RoboDK station: SpiralMeca.rdk

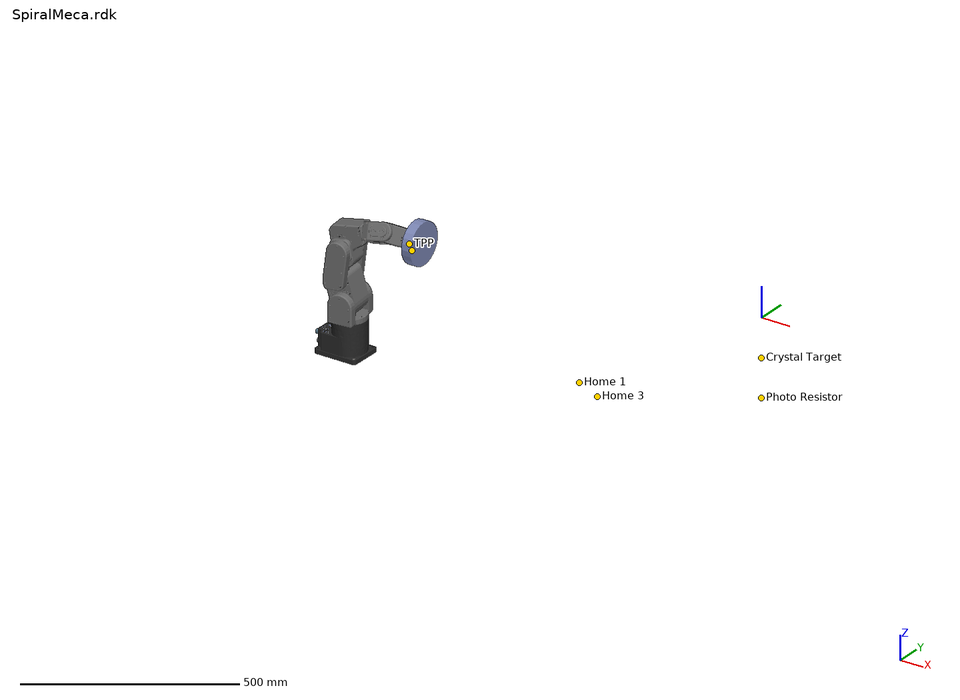
[picture v0: the station drawn from its stored meshes, robots at their saved joint values, targets as dots, program paths as lines]
Station SpiralMeca (saved by RoboDK 5.5.2). Poses are relative to the parent item; angles as X-Y-Z fixed-axis rotations.
  - robot Mecademic Meca500 R3: 6 axes
      modified DH rows (alpha deg, a mm, theta deg, d mm): 0, 0, 0, 135; -90, 0, -90, 0; 0, 135, 0, 0; -90, 38, 0, 120; 90, 0, 0, 0; -90, 0, 180, 70
      joint limits [-150, -70, -135, -170, -115, -720] to [150, 90, 70, 170, 115, 720]; home [0, 0, 0, 0, 0, 0]; saved at [5.545, -3.441, -6.55, -29.231, 11.413, 28.746]
    - tool CrystalToolSample, TCP at (0, 0, 0) mm, size 107.9 x 25.4 x 107.9 mm, geometry from CrystalToolSample.STEP
  - frame LED at (1143, 0, 409.6) mm
    - target TPP (Cartesian target) at (-970, -10, -81.6) mm, rotated rx 0 ry 90 rz 0 deg; joints [-5.545, -3.441, -6.55, 29.231, 11.413, -28.746] of Mecademic Meca500 R3
    - target Home 3 (Cartesian target) at (245.4, -1000, 268) mm, rotated rx 0 ry 90 rz 0 deg; joints [0, 10.295, 7.197, 0, -17.492, 0] of Mecademic Meca500 R3
    - target Home 1 (joint target) at (215.4, -1030, 308) mm, rotated rx 0 ry 90 rz 0 deg; joints [0, 0, 0, 0, 0, 0] of Mecademic Meca500 R3
    - target Target 47 (joint target) at (342.4, -1030, 308) mm, rotated rx 0 ry 90 rz 0 deg; joints [0, 11.211, -12.445, 0, 1.234, 0] of Mecademic Meca500 R3
    - target Photo Resistor (Cartesian target) at (0, 0, -203.2) mm; joints [0, 0, 0, 0, 0, 0] of Mecademic Meca500 R3
    - target Crystal Target (Cartesian target) at (0, 0, -101.6) mm; joints [-23.128, -26.053, 31.636, -77.168, -23.756, 166.237] of Mecademic Meca500 R3
    - target Target 7 (Cartesian target) at (-970.2, 0, -101.6) mm, rotated rx 0 ry 90 rz 0 deg; joints [0, -22.455, 17.494, 0, 4.961, 0] of Mecademic Meca500 R3
    - target Target 8 (Cartesian target) at (-970.2, 0, -101.6) mm, rotated rx 0 ry 90 rz 0 deg; joints [0, -33.951, 22.527, 0, 11.424, 0] of Mecademic Meca500 R3
  - Python program Spiral (listed below)
  - Python program Go Home (listed below)
  - Python program TEST SSAP (listed below)
  - Python program Prog4 (listed below)
  - Python program Linear Move (listed below)
  - Python program SSAP (listed below)
    - Python program Test SSAP 2 (listed below)
    - Python program Test SSAP 3 (listed below)
    - Python program Smart Spiral SSAP (listed below)
  - Python program Set Target Pos (listed below)
  - Python program Hexagon Test (listed below)
  - Python program Prog12 (listed below)
  - Python program Prog13 (listed below)

--- Python program Spiral ---
"""
Created on Thu Jan 19 18:43:18 2023

@author: westj
"""
from robodk.robolink import *       # import the robolink library (bridge with RoboDK)
RDK = Robolink()
from robodk.robomath import *
import math
import numpy as np
import matplotlib.pyplot as plt

class Spiral:
    def __init__(self,x0:float,y0:float,points:float) -> None:
        self.x0=x0 #x offset
        self.y0=y0 #y offset
        self.points=points

    def build(self, radius:float, spacing:float):
        revs=radius/spacing            #calc number of revolutions
        k=spacing/(2*np.pi)
        theta=np.array(np.linspace(0,revs*2*np.pi,self.points)) #how many points and angle coord
        r=k * theta                       #radius coord
        x=(r*np.cos(theta)+self.x0)
        y=(r*np.sin(theta)+self.y0)             #convert to y cartesian

        return x, y #convert to x cartesian


if __name__=="__main__":
    print('Calling spiral from class')
    R=30
    S=10
    TSpeed=10
    cur_spiral=Spiral(0,0,500)
    x,y=cur_spiral.build(R,S)


 #   print(cur_spiral.build(R,S))
  #  plt.plot(x, y, color = 'red', marker = "o")
  #  plt.axis('equal')
  #  plt.show()

#______Robot Movement_________________________________________

robot = RDK.Item('Mecademic Meca500 R3')
home = RDK.Item('Home 1')
target = RDK.Item('Target 2')# retrieve the Target item


robot.MoveJ(home)

robot.MoveJ(target)                 # move the robot to the target
#for i in x:
    #robot.MoveL(target.Pose()*transl(coord))

for i in range(len(x)):

    coord=(x[i],y[i],0)
    robot.MoveJ(target.Pose()*transl(coord))
    robot.WaitFinished()
    #print(coord)
    #print('')

--- Python program Go Home ---
# Type help("robodk.robolink") or help("robodk.robomath") for more information
# Press F5 to run the script
# Documentation: https://robodk.com/doc/en/RoboDK-API.html
# Reference:     https://robodk.com/doc/en/PythonAPI/robodk.html
# Note: It is not required to keep a copy of this file, your Python script is saved with your RDK project

# You can also use the new version of the API:
from robodk import robolink    # RoboDK API
from robodk import robomath    # Robot toolbox
RDK = robolink.Robolink()

robot = RDK.Item('Mecademic Meca500 R3')
home = RDK.Item('Home 1')
robot.MoveJ(home)

--- Python program TEST SSAP ---
"""
Created on Thu Jan 19 18:43:18 2023

@author: westj
"""
from robodk.robolink import *       # import the robolink library (bridge with RoboDK)
RDK = Robolink()
from robodk.robomath import *
import math
import numpy as np
import matplotlib.pyplot as plt
import array
import pandas as pd
from scipy.signal import find_peaks
from scipy.stats import linregress

class Spiral:
    def __init__(self,x0:float,y0:float,points:float) -> None:
        self.x0=x0 #x offset
        self.y0=y0 #y offset
        self.points=points

    def build(self, radius:float, spacing:float):
        revs=radius/spacing            #calc number of revolutions
        k=spacing/(2*np.pi)
        theta=np.array(np.linspace(0,revs*2*np.pi,self.points)) #how many points and angle coord
        r=k * theta                       #radius coord
        x=(r*np.cos(theta)+self.x0)       #convert to x cartesian
        y=(r*np.sin(theta)+self.y0)       #convert to y cartesian

        return x, y

class Linear:
    def __init__(self,data,points):
        self.data=data #data
        self.points=points #x offset

    def get(self,x):
        peaks= find_peaks(self.data['Intensity'], height=.1)

        H=peaks[1]['peak_heights']
        A=[]
        for i in range(len(IPeaks)):
            corr=[IPeaks[i],H[i]]
            A.append(corr)
        SA=sorted(A, key=lambda x: x[1], reverse=True) #sort by peak height largest to smallest
        print(SA)
        XPP=[]
        YPP=[]
        for i in range(self.points):
            #ICP.append(SA[i][0])
            XPP.append(self.data['X'][SA[i][0]])
            YPP.append(self.data['Y'][SA[i][0]])
        LRR=linregress(XPP,YPP)

        return LRR[0]*x+LRR[1]


class Intensity: #intensity function is a gaussian curve
    def __init__(self,x0:float,y0:float, mu_x, mu_y, sigma_x, sigma_y):
        self.x0=-x0 #x offset
        self.y0=-y0 #y offset
        self.mu_x=mu_x
        self.mu_y=mu_y
        self.sigma_x=sigma_x #x squish/stretch
        self.sigma_y=sigma_y #y sqush/stretch


    def get(self,x, y): #gaussian curve definition
        I=np.exp(-0.5 * (((x +self.x0- self.mu_x) / self.sigma_x)**2 + ((y+self.y0 - self.mu_y) / self.sigma_y)**2))
        return I


#*****************************************************************************************************************
#___Initialization______________
xl=0
yl=0
Loops=3
robot = RDK.Item('Mecademic Meca500 R3')
home = RDK.Item('Home 1')
target = RDK.Item('Target 2')# retrieve the Target item

robot.MoveJ(home)
robot.MoveJ(target)



for L in range(1,Loops+1):
    print(L)
    if __name__=="__main__":
        print('Calling spiral from class')

        cur_spiral=Spiral(xl,yl,200) #setting params of the spiral we will be using
        x,y=cur_spiral.build(10/L**L,5/L) #build our spiral x y coords
        Ix=1.24
        Iy=-2.3
        TestInt=Intensity(Ix,Iy,0,0,10,10) #set test intensity parameters

        #Plot our spiral
        # plt.plot(x, y, color = 'red', marker = "o")
        # plt.axis('equal')
        # plt.show()

    #initialize params
    X=[]
    Y=[]
    Z=[]
    Iv=[]
    Cv=[]

    for i in range(len(x)): #loop to get coord and corresponding intensity
        coord=(x[i],y[i],0)
        X.append(x[i])
        Y.append(y[i])
        Z.append(0)
        Ic=TestInt.get(x[i],y[i])
        Iv.append(np.array(Ic))

        robot.MoveJ(target.Pose()*transl(coord))
        robot.WaitFinished()
        #pandas dictionary
        titled_columns={'X': X,'Y': Y,'Z': Z,
                        'Intensity': Iv}
        data = pd.DataFrame(titled_columns)


    peaks= find_peaks(data['Intensity'], height=.1)
    IPeaks=peaks[0]
    H=peaks[1]['peak_heights']
    A=[]
    for i in range(len(IPeaks)):
        corr=[IPeaks[i],H[i]]
        A.append(corr)



    SA=sorted(A, key=lambda x: x[1], reverse=True) #sort by peak height largest to smallest
    if len(SA) == 1:
        print('one peak detected')
        break
    else:

     CL=Linear(data,2) #current linear line definition

    step=.1/L #linear step size
    xl=data['X'][SA[0][0]] #start x
    yl=CL.get(xl) #start y

    Xl=[xl]
    Yl=[yl]
    Il=[TestInt.get(xl,yl)]

    if  data['X'][SA[0][0]] < data['X'][SA[1][0]]:
        step=step
    else:
        step=-step


    while TestInt.get(xl+step,CL.get(xl+step)) >= TestInt.get(xl,CL.get(xl)):

        xl=xl+step
        yl=CL.get(xl)
        il=TestInt.get(xl,yl)
        Xl.append(xl)
        Yl.append(yl)
        Il.append(il)
        coord=(xl,yl,0)
        robot.MoveJ(target.Pose()*transl(coord))



    LLdata={'X':Xl,'Y':Yl,'I':Il}
    Ldata=pd.DataFrame(LLdata)

    fig = plt.figure()
    plt.style.use('seaborn-notebook')
    ax = fig.add_subplot(111, projection='3d')
    ax.plot3D(data['X'], data['Y'], data['Intensity'])
    ax.plot3D(data['X'][IPeaks], data['Y'][IPeaks], data['Intensity'][IPeaks],"x")
    ax.plot3D(Xl, Yl, Il,'o')

    ax.set_xlabel('X axis')
    ax.set_ylabel('Y axis')
    ax.set_zlabel('Z axis')
plt.show()




E=np.sqrt((Ix-xl)**2+(Iy-yl)**2)
print('***Linear Translation********************************************************')
print(Ldata)
print('_________SSAP Report:_________')
print('Calculated peak is at',xl,yl)
print('True peak is at',Ix,Iy)
print('Error is:',E)
print('Linear step size is:',step)

--- Python program Prog4 ---
# -*- coding: utf-8 -*-
"""
Created on Tue Feb 14 10:13:50 2023

@author: ChatGPT/ Jeremy West
"""

import math
from robodk.robolink import *
from robodk import robomath
RDK = Robolink()

target = RDK.Item('Target 2')# retrieve the Target item
robot = RDK.Item('Mecademic Meca500 R3')

# Define the position of the robot's tool
x = 100
y = 100
z = 300

# Define the orientation of the robot's tool using Euler angles (in degrees)
a = 0   # rotation around x-axis
b = 0    # rotation around y-axis
g = 0    # rotation around z-axis


# Set the robot's tool pose to the defined pose
#robodk.robomath.TxyzRxyz_2_Pose(xyzrpw) #[x,y,z,a,b,g]

#pose=robodk.robomath.Pose([x,y,z,a,b,g])
robot.setJoints([0,0,0,0,0,0])
robot.MoveJ(target)
approach = target.Pose()*transl(0,0,-100)
robot.MoveL(approach)

#print(pose)


robot.setPose(pose)

--- Python program Linear Move ---
from robodk.robolink import *       # import the robolink library (bridge with RoboDK)
from robodk.robomath import *       # import the robotics toolbox
RDK = Robolink()                    # establish a link with the simulator
robot = RDK.Item('Mecademic Meca500 R3')     # retrieve the robot by name


robot.setSpeed(100)  # Set linear speed in mm/s
robot.setJoints([0,0,0,0,0,0])      # set all robot axes to zero

tool=RDK.Item('CrystalToolSample')
robot.setPoseTool(tool) # Update the TCP

target = RDK.Item('TPP')         # retrieve the Target item
robot.MoveJ(target)                 # move the robot to the target


Final = target.Pose()*transl(0,20,0)
print(target.Pose())

rj=robot.Joints()

print(robot.MoveL_Test(rj,Final))

if robot.MoveL_Test(rj,Final) == 0:         # linear move to the approach position
    robot.MoveL(Final)


print('approach reached')
print('Attempting pose', Final)
#robot.MoveL(pose)

--- Python program SSAP ---
"""
Created on Thu Jan 19 18:43:18 2023

@author: westj
"""
from robodk.robolink import *       # import the robolink library (bridge with RoboDK)
RDK = Robolink()
from robodk.robomath import *
import math
import numpy as np
import matplotlib.pyplot as plt
import array
import pandas as pd
import requests
import re
from scipy.signal import find_peaks
from scipy.stats import linregress

class Spiral:
    def __init__(self,x0:float,y0:float,points:float) -> None:
        self.x0=x0 #x offset
        self.y0=y0 #y offset
        self.points=points

    def build(self, radius:float, spacing:float):
        revs=radius/spacing            #calc number of revolutions
        k=spacing/(2*np.pi)
        theta=np.array(np.linspace(0,revs*2*np.pi,self.points)) #how many points and angle coord
        r=k * theta                       #radius coord
        x=(r*np.cos(theta)+self.x0)       #convert to x cartesian
        y=(r*np.sin(theta)+self.y0)       #convert to y cartesian

        return x, y

class Linear:
    def __init__(self,data,points):
        self.data=data #data
        self.points=points #x offset

    def get(self,x):
        peaks= find_peaks(self.data['Intensity'], height=-900)

        H=peaks[1]['peak_heights']
        A=[]
        for i in range(len(IPeaks)):
            corr=[IPeaks[i],H[i]]
            A.append(corr)
        SA=sorted(A, key=lambda x: x[1], reverse=True) #sort by peak height largest to smallest
        print(SA)
        XPP=[]
        YPP=[]
        for i in range(self.points):
            #ICP.append(SA[i][0])
            XPP.append(self.data['X'][SA[i][0]])
            YPP.append(self.data['Y'][SA[i][0]])
        LRR=linregress(XPP,YPP)

        return LRR[0]*x+LRR[1]


class Intensity: #intensity function is a gaussian curve
    def __init__(self,x0:float,y0:float, mu_x, mu_y, sigma_x, sigma_y):
        self.x0=-x0 #x offset
        self.y0=-y0 #y offset
        self.mu_x=mu_x
        self.mu_y=mu_y
        self.sigma_x=sigma_x #x squish/stretch
        self.sigma_y=sigma_y #y sqush/stretch


    def get(self,x, y): #gaussian curve definition
        I=np.exp(-0.5 * (((x +self.x0- self.mu_x) / self.sigma_x)**2 + ((y+self.y0 - self.mu_y) / self.sigma_y)**2))
        return I

class Photoresistor:
    def __init__(self,url) -> None:
        self.url=url
    def get(self):
        response = requests.get(self.url)
        if response.ok:
            value = response.text
            pr=re.findall(r'\d+',value)
            pri=-int(pr[0])
            #print('Received value:', value)
            #print('Number', PR)
        else:
            print('Error:', response.status_code)


        return pri


#*****************************************************************************************************************
#___Initialization______________
xl=0
yl=0
Loops=3
robot = RDK.Item('Mecademic Meca500 R3')
home = RDK.Item('Home 1')
target = RDK.Item('Target 2')# retrieve the Target item
PR=Photoresistor( 'http://192.168.0.24')

robot.MoveJ(home)
robot.MoveJ(target)



for L in range(1,Loops+1):
    print(L)
    if __name__=="__main__":
        print('Calling spiral from class')

        cur_spiral=Spiral(xl,yl,200) #setting params of the spiral we will be using
        x,y=cur_spiral.build(30/L**L,5/L) #build our spiral x y coords
        Ix=1.24
        Iy=-2.3
        TestInt=Intensity(Ix,Iy,0,0,10,10) #set test intensity parameters

        #Plot our spiral
        # plt.plot(x, y, color = 'red', marker = "o")
        # plt.axis('equal')
        # plt.show()

    #initialize params
    X=[]
    Y=[]
    Z=[]
    Iv=[]
    Cv=[]

    for i in range(len(x)): #loop to get coord and corresponding intensity
        coord=(x[i],y[i],0)
        X.append(x[i])
        Y.append(y[i])
        Z.append(0)
        Ic=PR.get()

        Iv.append(np.array(Ic))

        robot.MoveJ(target.Pose()*transl(coord))
        robot.WaitFinished()
        #pandas dictionary
        titled_columns={'X': X,'Y': Y,'Z': Z,
                        'Intensity': Iv}
        data = pd.DataFrame(titled_columns)


    peaks= find_peaks(data['Intensity'], height=-900)
    print('peaks',peaks)


    IPeaks=peaks[0]
    H=peaks[1]['peak_heights']
    A=[]
    for i in range(len(IPeaks)):
        corr=[IPeaks[i],H[i]]

        A.append(corr)



    SA=sorted(A, key=lambda x: x[1], reverse=True) #sort by peak height largest to smallest
    if len(SA) == 1:
        print('one peak detected')
        break
    else:

     CL=Linear(data,2) #current linear line definition

    step=.1/L #linear step size
    xl=data['X'][SA[0][0]] #start x
    yl=CL.get(xl) #start y

    Xl=[xl]
    Yl=[yl]
    PRS=SA[0][1]
    Il=[PRS]

    if  data['X'][SA[0][0]] < data['X'][SA[1][0]]:
        step=step
    else:
        step=-step


    while PR.get() >= .99*PRS:

        xl=xl+step
        yl=CL.get(xl)
        PRS=PR.get()
        Xl.append(xl)
        Yl.append(yl)
        Il.append(PRS)
        coord=(xl,yl,0)
        robot.MoveJ(target.Pose()*transl(coord))



    LLdata={'X':Xl,'Y':Yl,'I':Il}
    Ldata=pd.DataFrame(LLdata)

    fig = plt.figure()
    plt.style.use('seaborn-notebook')
    ax = fig.add_subplot(111, projection='3d')
    ax.plot3D(data['X'], data['Y'], data['Intensity'])
    ax.plot3D(data['X'][IPeaks], data['Y'][IPeaks], data['Intensity'][IPeaks],"x")
    ax.plot3D(Xl, Yl, Il,'o')

    ax.set_xlabel('X axis')
    ax.set_ylabel('Y axis')
    ax.set_zlabel('Z axis')
plt.show()




E=np.sqrt((Ix-xl)**2+(Iy-yl)**2)
print('***Linear Translation********************************************************')
print(Ldata)
print('_________SSAP Report:_________')
print('Calculated peak is at',xl,yl)
print('True peak is at',Ix,Iy)
print('Error is:',E)
print('Linear step size is:',step)

--- Python program Test SSAP 2 ---
"""
Created on Thu Jan 19 18:43:18 2023

@author: westj
"""
from robodk.robolink import *       # import the robolink library (bridge with RoboDK)
RDK = Robolink()
from robodk.robomath import *
import math
import numpy as np
import matplotlib.pyplot as plt
import array
import pandas as pd
import requests
import re
from scipy.signal import find_peaks
from scipy.stats import linregress
#******CLASSES AND CLASS FUNCTIONS****************************************************************************
class Spiral:
    def __init__(self,x0:float,y0:float,points:float) -> None:
        self.x0=x0 #x offset
        self.y0=y0 #y offset
        self.points=points

    def build(self, radius:float, spacing:float):
        revs=radius/spacing            #calc number of revolutions
        k=spacing/(2*np.pi)
        theta=np.array(np.linspace(0,revs*2*np.pi,self.points)) #how many points and angle coord
        r=k * theta                       #radius coord
        x=(r*np.cos(theta)+self.x0)       #convert to x cartesian
        y=(r*np.sin(theta)+self.y0)       #convert to y cartesian
        return x, y

class Linear:
    def __init__(self,data,points):
        self.data=data #data
        self.points=points #x offset

    def get(self,x):
        peaks= find_peaks(self.data['Intensity'], height=-900)
        IPeaks=peaks[0]
        H=peaks[1]['peak_heights']
        A=[]
        for i in range(len(IPeaks)):
            corr=[IPeaks[i],H[i]]
            A.append(corr)
        SA=sorted(A, key=lambda x: x[1], reverse=True) #sort by peak height largest to smallest
        if len(SA) <= 1:

            E=np.sqrt((Ix-xl)**2+(Iy-yl)**2)
            print('***Linear Translation********************************************************')
            print(Ldata)
            print('_________SSAP Report:_________')
            print('Calculated peak is at',xl,yl)
            print('True peak is at',Ix,Iy)
            print('Error is:',E)
            print('Linear step size is:',step)
            raise Exception("Spiral did not find enough peaks")
        XPP=[]
        YPP=[]
        for i in range(self.points):
            #ICP.append(SA[i][0])
            XPP.append(self.data['X'][SA[i][0]])
            YPP.append(self.data['Y'][SA[i][0]])
        LRR=linregress(XPP,YPP)

        return LRR[0]*x+LRR[1]

    def getSA(self):
        peaks= find_peaks(self.data['Intensity'], height=-900)
        IPeaks=peaks[0]
        H=peaks[1]['peak_heights']
        A=[]
        for i in range(len(IPeaks)):
            corr=[IPeaks[i],H[i]]
            A.append(corr)
        SA=sorted(A, key=lambda g: g[1], reverse=True) #sort by peak height largest to smallest
        return SA,IPeaks

class Intensity: #intensity function is a gaussian curve
    def __init__(self,x0:float,y0:float, mu_x, mu_y, sigma_x, sigma_y):
        self.x0=-x0 #x offset
        self.y0=-y0 #y offset
        self.mu_x=mu_x
        self.mu_y=mu_y
        self.sigma_x=sigma_x #x squish/stretch
        self.sigma_y=sigma_y #y sqush/stretch


    def get(self,x, y): #gaussian curve definition
        I=np.exp(-0.5 * (((x +self.x0- self.mu_x) / self.sigma_x)**2 + ((y+self.y0 - self.mu_y) / self.sigma_y)**2))
        return I

class Photoresistor:
    def __init__(self,url) -> None:
        self.url=url
    def get(self):
        response = requests.get(self.url)
        if response.ok:
            value = response.text
            pr=re.findall(r'\d+',value)
            pri=-int(pr[0])
            #print('Received value:', value)
            #print('Number', PR)
        else:
            print('Error:', response.status_code)


        return pri


#***SPIRAL SCANNING ALIGNMENT PROCEDURE**************************************************************************************************************
#___Initialization______________
xl=0 #starting offset from target for spiral
yl=0
Loops=2 #number of loops to run SSAP

robot = RDK.Item('Mecademic Meca500 R3') #define robot
home = RDK.Item('Home 1') #define robot home
target = RDK.Item('Target 2')# retrieve the Target item
PR=Photoresistor( 'http://192.168.0.24') #Photoresistor webserver IP

robot.MoveJ(home)
print('Robot homed')
robot.MoveJ(target)
print('Robot target approached')

for L in range(1,Loops+1):
    if __name__=="__main__":
        print('Starting Spiral '+str(L))

        cur_spiral=Spiral(xl,yl,200) #setting params of the spiral we will be using
        x,y=cur_spiral.build(20/L**L,3/L) #build our spiral x y coords
        Ix=-15.24
        Iy=25.3
        TestInt=Intensity(Ix,Iy,0,0,10,10) #set test intensity parameters

        #Plot our spiral
        # plt.plot(x, y, color = 'red', marker = "o")
        # plt.axis('equal')
        # plt.show()

    #initialize params
    X=[]
    Y=[]
    Z=[]
    Iv=[]
    Cv=[]

    for i in range(len(x)): #loop to get coord and corresponding intensity
        coord=(x[i],y[i],0)
        X.append(x[i])
        Y.append(y[i])
        Z.append(0)
        #Ic=PR.get() #get intensity for PR for online run
        Ic=TestInt.get(x[i],y[i]) #test intensity get
        Iv.append(np.array(Ic))

        robot.MoveJ(target.Pose()*transl(coord))
        robot.WaitFinished()

        #pandas dictionary
        titled_columns={'X': X,'Y': Y,'Z': Z,
                        'Intensity': Iv}
        data = pd.DataFrame(titled_columns)

    print('Spiral ' +str(L)+ ' Completed')

    CL=Linear(data,2) #current linear line definition
    SA,IPeaks=CL.getSA()

    step=.1/L #linear step size
    xl=data['X'][SA[0][0]] #start x
    yl=CL.get(xl) #start y

    Xl=[xl,xl,xl]
    Yl=[yl,yl,yl]
    PRS=SA[0][1]
    Il=[PRS,PRS,PRS]
    ave_c=3 #number of intetensity terms to average
    IAv=np.average(Il[:ave_c])

    if  data['X'][SA[0][0]] < data['X'][SA[1][0]]:  #find direction to move based on location of next highest intensity
        step=-step
    else:
        step=step

    print('Linear move '+str(L)+ ': STARTED')
    while PRS >= .99*IAv:
        IAv=np.average(Il[:ave_c])
        xl=xl+step
        yl=CL.get(xl)
        #PRS=PR.get()
        PRS=TestInt.get(xl,yl)
        Xl.append(xl)
        Yl.append(yl)
        Il.append(PRS)
        coord=(xl,yl,0)
        robot.MoveJ(target.Pose()*transl(coord))
    print('Linear move '+str(L)+ ': COMPLETED')

    LLdata={'X':Xl,'Y':Yl,'I':Il}
    Ldata=pd.DataFrame(LLdata)

    Lmax_I=Il.index(max(Ldata['I']))
    xl=Xl[Lmax_I]
    yl=Yl[Lmax_I]

    fig = plt.figure()
    #plt.style.use('seaborn-notebook')
    ax = fig.add_subplot(111, projection='3d')
    ax.plot3D(data['X'], data['Y'], data['Intensity'])
    ax.plot3D(data['X'][IPeaks], data['Y'][IPeaks], data['Intensity'][IPeaks],"x")
    ax.plot3D(xl, yl, max(Ldata['I']),"x")
    ax.plot3D(Xl, Yl, Il,'o')

    ax.set_xlabel('X axis')
    ax.set_ylabel('Y axis')
    ax.set_zlabel('Z axis')
plt.show()




E=np.sqrt((Ix-xl)**2+(Iy-yl)**2)
print('***Linear Translation********************************************************')
print(Ldata)
print('_________SSAP Report:_________')
print('Calculated peak is at',xl,yl)
print('True peak is at',Ix,Iy)
print('Error is:',E)
print('Linear step size is:',step)

--- Python program Test SSAP 3 ---
"""
Created on Thu Jan 19 18:43:18 2023

@author: westj
"""
from robodk.robolink import *       # import the robolink library (bridge with RoboDK)
RDK = Robolink()
from robodk.robomath import *
import math
import numpy as np
import matplotlib.pyplot as plt
import array
import pandas as pd
import requests
import re
from scipy.signal import find_peaks, peak_prominences
from scipy.stats import linregress
#******CLASSES AND CLASS FUNCTIONS****************************************************************************
class Spiral:
    def __init__(self,x0:float,y0:float,points:float) -> None:
        self.x0=x0 #x offset
        self.y0=y0 #y offset
        self.points=points

    def build(self, radius:float, spacing:float):
        revs=radius/spacing            #calc number of revolutions
        k=spacing/(2*np.pi)
        theta=np.array(np.linspace(0,revs*2*np.pi,self.points)) #how many points and angle coord
        r=k * theta                       #radius coord
        x=(r*np.cos(theta)+self.x0)       #convert to x cartesian
        y=(r*np.sin(theta)+self.y0)       #convert to y cartesian
        return x, y

class Linear:
    def __init__(self,data,points):
        self.data=data #data
        self.points=points #number of points to fit

    def get(self,x):
        peaks= find_peaks(self.data['Intensity'], height=-900)
        IPeaks=peaks[0]
        H=peaks[1]['peak_heights']
        A=[]
        for i in range(len(IPeaks)):
            corr=[IPeaks[i],H[i]]
            A.append(corr)
        SA=sorted(A, key=lambda x: x[1], reverse=True) #sort by peak height largest to smallest
        if len(SA) <= 1:

            E=np.sqrt((Ix-xl)**2+(Iy-yl)**2)
            print('***Linear Translation********************************************************')
            print(Ldata)
            print('_________SSAP Report:_________')
            print('Calculated peak is at',xl,yl)
            print('True peak is at',Ix,Iy)
            print('Error is:',E)
            print('Linear step size is:',step)
            raise Exception("Spiral did not find enough peaks")
        XPP=[]
        YPP=[]
        for i in range(self.points):
            #ICP.append(SA[i][0])
            XPP.append(self.data['X'][SA[i][0]])
            YPP.append(self.data['Y'][SA[i][0]])
        LRR=linregress(XPP,YPP)

        return LRR[0]*x+LRR[1]
    def getC(self,x,xl,yl):
        peaks= find_peaks(self.data['Intensity'], prominence=[.1],width=3) #find peaks
        XPP=[xl]  #use origin of previous spiral as a point
        YPP=[yl]
        XPP.append(self.data['X'][peaks[0][0]])
        YPP.append(self.data['Y'][peaks[0][0]])
        LRR=linregress(XPP,YPP) #run regression
        return LRR[0]*x+LRR[1]


    def getSA(self):
        peaks= find_peaks(self.data['Intensity'], prominence=[.1],width=3)
        IPeaks=peaks[0]
        H=peaks[1]['peak_heights']
        A=[]
        for i in range(len(IPeaks)):
            corr=[IPeaks[i],H[i]]
            A.append(corr)
        SA=sorted(A, key=lambda g: g[1], reverse=True) #sort by peak height largest to smallest
        return SA,IPeaks

class Intensity: #intensity function is a gaussian curve
    def __init__(self,x0:float,y0:float, mu_x, mu_y, sigma_x, sigma_y):
        self.x0=-x0 #x offset
        self.y0=-y0 #y offset
        self.mu_x=mu_x
        self.mu_y=mu_y
        self.sigma_x=sigma_x #x squish/stretch
        self.sigma_y=sigma_y #y sqush/stretch


    def get(self,x, y): #gaussian curve definition
        I=np.exp(-0.5 * (((x +self.x0- self.mu_x) / self.sigma_x)**2 + ((y+self.y0 - self.mu_y) / self.sigma_y)**2))
        return I

class Photoresistor:
    def __init__(self,url) -> None:
        self.url=url
    def get(self):
        response = requests.get(self.url)
        if response.ok:
            value = response.text
            pr=re.findall(r'\d+',value)
            pri=-int(pr[0])
            #print('Received value:', value)
            #print('Number', PR)
        else:
            print('Error:', response.status_code)


        return pri


#***SPIRAL SCANNING ALIGNMENT PROCEDURE**************************************************************************************************************
#___Initialization______________
xl=0 #starting offset from target for spiral
yl=0
Loops=4 #number of loops to run SSAP

robot = RDK.Item('Mecademic Meca500 R3') #define robot
home = RDK.Item('Home 1') #define robot home
target = RDK.Item('Target 2')# retrieve the Target item
PR=Photoresistor( 'http://192.168.0.24') #Photoresistor webserver IP

robot.MoveJ(home)
print('Robot homed')
robot.MoveJ(target)
print('Robot target approached')

for L in range(1,Loops+1):
    if __name__=="__main__":
        print('Starting Spiral '+str(L))

        cur_spiral=Spiral(xl,yl,200) #setting params of the spiral we will be using
        revs=20/L**L/3/L
        points=200
        x,y=cur_spiral.build(30/L**L,3/L**2) #build our spiral x y coords
        Ix=-10
        Iy=10
        TestInt=Intensity(Ix,Iy,0,0,10,10) #set test intensity parameters


        #Plot our spiral
        # plt.plot(x, y, color = 'red', marker = "o")
        # plt.axis('equal')
        # plt.show()

    #initialize params
    X=[]
    Y=[]
    Z=[]
    Iv=[]
    Cv=[]
    #while loop here instead or an if thing with a point at 0,0,0 need to make a new linear fit function maybe or pass it different args
    for i in range(1,len(x)): #loop to get coord and corresponding intensity
        if not find_peaks(Iv,prominence=[.1],width=3)[0]: #check if we found a peak
            coord=(x[i],y[i],0)
            X.append(x[i])
            Y.append(y[i])
            Z.append(0)
            #Ic=PR.get() #get intensity for PR for online run
            Ic=TestInt.get(x[i],y[i]) #test intensity get
            Iv.append(np.array(Ic))

            robot.MoveJ(target.Pose()*transl(coord))
            robot.WaitFinished()
        else:
            ps=find_peaks(Iv,prominence=[.1],width=3)[0][0]
            print(ps)
            fig1 = plt.figure()
            #plt.style.use('seaborn-notebook')
            theta=np.array(np.linspace(0,revs*2*np.pi,points))
            peaks, _ = find_peaks(Iv)

            # height=.1,distance=3,threshold=0.01,
            prominences = peak_prominences(Iv, peaks)[0]
            contour_heights = np.array(Iv)[peaks] - prominences
            plt.plot(Iv)
            plt.plot(peaks, np.array(Iv)[peaks], "x")
            plt.vlines(x=peaks, ymin=contour_heights, ymax=np.array(Iv)[peaks])
            plt.show()

            fig = plt.figure()



            ax = fig.add_subplot(111, projection='3d')
            ax.plot3D(X, Y, Iv)
            ax.plot3D(X[ps], Y[ps], Iv[ps],'x')



            ax.set_xlabel('X axis')
            ax.set_ylabel('Y axis')
            ax.set_zlabel('Z axis')
            plt.show()
            break

    print('peak',find_peaks(Iv,prominence=[.1],width=3)[0])
    print('length',len(find_peaks(Iv,prominence=[.1],width=3)[0]))

    #pandas dictionary
    titled_columns={'X': X,'Y': Y,'Z': Z,
                        'Intensity': Iv}
    data = pd.DataFrame(titled_columns)
    print('Spiral ' +str(L)+ ' Completed')

    CL=Linear(data,2) #current linear line definition
    #SA,IPeaks=CL.getSA()



    step=.1/L #linear step size


    peaks= find_peaks(data['Intensity'],height=-900,prominence=[.1],width=3)

    IPeaks=peaks[0][0]


    xL=data['X'][IPeaks]
    yL=CL.getC(xL,xl,yl) #start y

    Xl=[xL]
    Yl=[yL]

    PRS=data['Intensity'][IPeaks]
    Il=[PRS]

    if  data['X'][IPeaks] > 0:  #find direction to move
        step=step
    else:
        step=-step

    print('Linear move '+str(L)+ ': STARTED')


    while not find_peaks(Il,prominence=[.1],width=3)[0]: #linear move
        if max(Il) <= PRS:
            xL=xL+step
            yL=CL.getC(xL,xl,yl)
            #PRS=PR.get()
            PRS=TestInt.get(xL,yL)
            Xl.append(xL)
            Yl.append(yL)
            Il.append(PRS)
            coord=(xL,yL,0)
            robot.MoveJ(target.Pose()*transl(coord))

        else:
            break
    print('Linear move '+str(L)+ ': COMPLETED')

    LLdata={'X':Xl,'Y':Yl,'I':Il}
    Ldata=pd.DataFrame(LLdata)

    Lmax_I=Il.index(max(Ldata['I']))
    xl=Xl[Lmax_I]
    yl=Yl[Lmax_I]

    fig = plt.figure()
    #plt.style.use('seaborn-notebook')
    ax = fig.add_subplot(111, projection='3d')
    ax.plot3D(data['X'], data['Y'], data['Intensity'])
    ax.plot3D(data['X'][IPeaks], data['Y'][IPeaks], data['Intensity'][IPeaks],"x")
    ax.plot3D(xl, yl, max(Ldata['I']),"x")
    ax.plot3D(Xl, Yl, Il,'o')

    ax.set_xlabel('X axis')
    ax.set_ylabel('Y axis')
    ax.set_zlabel('Z axis')


    points=100
    xv,yv=np.meshgrid(np.linspace(-20,20,points),np.linspace(-20,20,points))
    iv=TestInt.get(xv,yv)
    ax.plot_surface(xv,yv,iv,alpha=0.5)
    plt.show()



E=np.sqrt((Ix-xl)**2+(Iy-yl)**2)
print('***Linear Translation********************************************************')
print(Ldata)
print('_________SSAP Report:_________')
print('Calculated peak is at',xl,yl)
print('True peak is at',Ix,Iy)
print('Error is:',E)
print('Linear step size is:',step)

--- Python program Smart Spiral SSAP ---
"""
Created on Thu Jan 19 18:43:18 2023

@author: westj
"""
from robodk.robolink import *       # import the robolink library (bridge with RoboDK)
RDK = Robolink()
from robodk.robomath import *
import math
import numpy as np
import matplotlib.pyplot as plt
import array
import pandas as pd
import requests
import re
from scipy.signal import find_peaks, peak_prominences, savgol_filter
from scipy.stats import linregress
#******CLASSES AND CLASS FUNCTIONS****************************************************************************
class Spiral:
    def __init__(self,x0:float,y0:float,points:float) -> None:
        self.x0=x0 #x offset
        self.y0=y0 #y offset
        self.points=points

    def build(self, radius:float, spacing:float):
        revs=radius/spacing            #calc number of revolutions
        k=spacing/(2*np.pi)
        theta=np.array(np.linspace(0,revs*2*np.pi,self.points)) #how many points and angle coord
        r=k * theta                       #radius coord
        x=(r*np.cos(theta)+self.x0)       #convert to x cartesian
        y=(r*np.sin(theta)+self.y0)       #convert to y cartesian
        return x, y

class Linear:
    def __init__(self,data,points):
        self.data=data #data
        self.points=points #number of points to fit

    def get(self,x):
        peaks= find_peaks(self.data['Intensity'], prominence=[prominence],width=width,height=height)
        IPeaks=peaks[0]
        H=peaks[1]['peak_heights']
        A=[]
        for i in range(len(IPeaks)):
            corr=[IPeaks[i],H[i]]
            A.append(corr)
        SA=sorted(A, key=lambda x: x[1], reverse=True) #sort by peak height largest to smallest
        if len(SA) <= 1:

            E=np.sqrt((Ix-xl)**2+(Iy-yl)**2)
            print('***Linear Translation********************************************************')
            print(Ldata)
            print('_________SSAP Report:_________')
            print('Calculated peak is at',xl,yl)
            print('True peak is at',Ix,Iy)
            print('Error is:',E)
            print('Linear step size is:',step)
            raise Exception("Spiral did not find enough peaks")
        XPP=[]
        YPP=[]
        for i in range(self.points):
            #ICP.append(SA[i][0])
            XPP.append(self.data['X'][SA[i][0]])
            YPP.append(self.data['Y'][SA[i][0]])
        LRR=linregress(XPP,YPP)

        return LRR[0]*x+LRR[1]
    def getC(self,x,xl,yl):
        peaks= find_peaks(self.data['Intensity'], prominence=[prominence],width=width,height=height) #find peaks
        XPP=[xl]  #use origin of previous spiral as a point
        YPP=[yl]
        XPP.append(self.data['X'][peaks[0][0]])
        YPP.append(self.data['Y'][peaks[0][0]])
        LRR=linregress(XPP,YPP) #run regression
        return LRR[0]*x+LRR[1]


    def getSA(self):
        peaks= find_peaks(self.data['Intensity'],prominence=[prominence],width=width,height=height)
        IPeaks=peaks[0]
        H=peaks[1]['peak_heights']
        A=[]
        for i in range(len(IPeaks)):
            corr=[IPeaks[i],H[i]]
            A.append(corr)
        SA=sorted(A, key=lambda g: g[1], reverse=True) #sort by peak height largest to smallest
        return SA,IPeaks

class Intensity: #intensity function is a gaussian curve
    def __init__(self,x0:float,y0:float, mu_x, mu_y, sigma_x, sigma_y):
        self.x0=-x0 #x offset
        self.y0=-y0 #y offset
        self.mu_x=mu_x
        self.mu_y=mu_y
        self.sigma_x=sigma_x #x squish/stretch
        self.sigma_y=sigma_y #y sqush/stretch


    def get(self,x, y): #gaussian curve definition
        I=np.exp(-0.5 * (((x +self.x0- self.mu_x) / self.sigma_x)**2 + ((y+self.y0 - self.mu_y) / self.sigma_y)**2))
        return I

class Photoresistor:
    def __init__(self,url) -> None:
        self.url=url
    def get(self):
        response = requests.get(self.url) #go to webserver under the url of the arduino/photoresistor
        if response.ok: #if we can connect
            value = response.text #screen scrape the web server
            pr=re.findall(r'\d+',value) #take the number off the webserver
            pri=-int(pr[0]) #reverse the sign of the number
            #print('Received value:', value)
            #print('Number', PR)
        else:
            print('Error:', response.status_code)


        return pri

#def Exit_SSAP(Intensity,plateau_size,height):
 #   if len(find_peaks(Intensity,plateau_size=pleatau_size,height=height)[0])>0:
    #    break

#***SPIRAL SCANNING ALIGNMENT PROCEDURE**************************************************************************************************************
#___Initialization______________
xl=0 #starting offset from target for spiral
yl=0
zl=0
Loops=3 #number of loops to run SSAP

robot = RDK.Item('Mecademic Meca500 R3') #define robot
home = RDK.Item('Home 1') #define robot home
target = RDK.Item('TPP')# retrieve the Target item
PR=Photoresistor( 'http://192.168.0.24') #Photoresistor webserver IP

robot.setSpeed(-1,75)
robot.MoveJ(home)
print('Robot homed')
robot.MoveJ(target)
print('Robot target approached')

for L in range(1,Loops+1):
    if __name__=="__main__":
        print('Starting Spiral '+str(L))

        cur_spiral=Spiral(xl,yl,300) #setting params of the spiral we will be using
        revs=20/L**L/3/L
        points=200
        x,y=cur_spiral.build(30/L**2,3/L**2) #build our spiral x y coords
        step=.01/L #linear step size
        zstep=2/L

        Ix=-10
        Iy=10
        TestInt=Intensity(Ix,Iy,0,0,10,10) #set test intensity parameters
        prominence=100
        width=3
        height=-900
        plateau_size=3 ############################################
        IAS=10


        #Plot our spiral
        # plt.plot(x, y, color = 'red', marker = "o")
        # plt.axis('equal')
        # plt.show()

    #initialize params
    X=[]
    Y=[]
    Z=[]
    Iv=[]
    Cv=[]

    for i in range(1,len(x)): #loop to get coord and corresponding intensity
        if len(find_peaks(Iv,prominence=[prominence],width=width,height=height)[0])<=0: #check if we found a peak
            if i==len(x):
                print('No peaks found in spiral: Spiral centered')
                coord=(xl,yl,zl)
                robot.MoveJ(target.Pose()*transl(coord))
                raise Exception('Alignment Acheived')
                break
            coord=(x[i],y[i],zl)
            X.append(x[i])
            Y.append(y[i])
            Z.append(0)
            Ic=PR.get() #get intensity for PR for online run
            #Ic=TestInt.get(x[i],y[i]) #test intensity get
            Iv.append(np.array(Ic))

            robot.MoveJ(target.Pose()*transl(coord))
            robot.WaitFinished()
        else:
            ps=find_peaks(Iv,prominence=[prominence],width=width,height=height)[0][0]
            fig1 = plt.figure()
            #plt.style.use('seaborn-notebook')
            theta=np.array(np.linspace(0,revs*2*np.pi,points))
            peaks, _ = find_peaks(Iv)

            # height=.1,distance=3,threshold=0.01,
            prominences = peak_prominences(Iv, peaks)[0]
            contour_heights = np.array(Iv)[peaks] - prominences
            plt.plot(Iv)
            plt.plot(peaks, np.array(Iv)[peaks], "x")
            plt.vlines(x=peaks, ymin=contour_heights, ymax=np.array(Iv)[peaks])
            plt.show()

            fig = plt.figure()

            ax = fig.add_subplot(111, projection='3d')
            ax.plot3D(X, Y, Iv)
            ax.plot3D(X[ps], Y[ps], Iv[ps],'x')

            ax.set_xlabel('X axis')
            ax.set_ylabel('Y axis')
            ax.set_zlabel('Z axis')
            plt.show()
            break


    #pandas dictionary
    titled_columns={'X': X,'Y': Y,'Z': Z,
                        'Intensity': Iv}
    data = pd.DataFrame(titled_columns)
    print('Spiral ' +str(L)+ ' Completed')

    if len(find_peaks(data['Intensity'],plateau_size=plateau_size,height=height)[0])>0: #check to see if we are at the peak
        PI=find_peaks(data['Intensity'],plateau_size=plateau_size,height=height)[0]
        xl=data['X'][PI]
        yl=data['Y'][PI]
        coord=(xl,yl,zl)
        robot.MoveJ(target.Pose()*transl(coord))
        print('SSAP Complete!')

        break



    CL=Linear(data,2) #current linear line definition


    peaks= find_peaks(data['Intensity'],height=height,prominence=[prominence],width=width)
    IPeaks=peaks[0][0]
    IPeaks=Iv.index(max(Iv))

    xL=data['X'][IPeaks]
    yL=CL.getC(xL,xl,yl) #start y

    Xl=[xL]
    Yl=[yL]

    PRS=data['Intensity'][IPeaks]
    Il=[PRS]

    if  data['X'][IPeaks] > xl:  #find direction to move
        step=step
    else:
        step=-step

    print('Linear move '+str(L)+ ': STARTED')

    #Linear search
    while len(find_peaks(Il,prominence=[prominence],width=width,height=height)[0])<=0: #linear move
        xL=xL+step
        yL=CL.getC(xL,xl,yl)
        PRLT=[]
        for j in range(IAS):
            PRL=PR.get()
            PRLT.append(PRL)

        LI=np.average(PRLT)
        print(PRLT)
        print(LI)
        #PRS=TestInt.get(xL,yL)
        Xl.append(xL)
        Yl.append(yL)
        Il.append(LI)
        print(LI)
        coord=(xL,yL,zl)
        robot.MoveJ(target.Pose()*transl(coord))

        #if len(find_peaks(-np.array(Il),plateau_size=4,prominence=30)[0])<=0:
        #    print('Linear moved past alignment')
        #    break

    print('Linear move '+str(L)+ ': COMPLETED')

    LLdata={'X':Xl,'Y':Yl,'I':Il}
    Ldata=pd.DataFrame(LLdata)

    Lmax_I=Il.index(max(Ldata['I']))
    xl=Xl[Lmax_I]
    yl=Yl[Lmax_I]

    fig = plt.figure()
    #plt.style.use('seaborn-notebook')
    ax = fig.add_subplot(111, projection='3d')
    ax.plot3D(data['X'], data['Y'], data['Intensity'])
    ax.plot3D(data['X'][IPeaks], data['Y'][IPeaks], data['Intensity'][IPeaks],"x")
    ax.plot3D(xl, yl, max(Ldata['I']),"x")
    ax.plot3D(Xl, Yl, Il,'o')

    ax.set_xlabel('X axis')
    ax.set_ylabel('Y axis')
    ax.set_zlabel('Z axis')
    plt.show()

    if len(find_peaks(Ldata['I'],plateau_size=plateau_size,height=height)[0])>0: #check to see if we are at the peak
        PI=find_peaks(Ldata['I'],plateau_size=plateau_size,height=height)[0]
        xl=Ldata['X'][PI]
        yl=Ldata['Y'][PI]
        coord=(xl,yl,zl)
        robot.MoveJ(target.Pose()*transl(coord))
        print('SSAP Complete!')
        break


    #Push Pull Search
    IPP=[]
    ZLPP=[]

    for i in range(3):
        coord=(xl,yl,zl)
        ZLPP.append(zl)
        robot.MoveJ(target.Pose()*transl(coord))
        PRPPT=[]
        for j in range(IAS):
            PRPP=PR.get()
            PRPPT.append(PRPP)
        PPI=np.average(PRPPT)
        IPP.append(PPI)

        zl=zl+(zstep)

    plt.plot(ZLPP,IPP)
    plt.show()

    if IPP.index(max(IPP))>0:
        zstep=zstep
    else:
        zstep=-zstep
    ZLPP=[]
    IPP=[]

    coord=(xl,yl,zl)
    robot.MoveJ(target.Pose()*transl(coord))
    #maybe savitzky golay or moving average filter
    while len(find_peaks(IPP,prominence=5,height=height)[0])<=0: #Push pull
        coord=(xl,yl,zl)
        ZLPP.append(zl)
        robot.MoveJ(target.Pose()*transl(coord))
        PRPPT=[]
        for j in range(IAS):
            PRPP=PR.get()
            PRPPT.append(PRPP)
        PPI=np.average(PRPPT)
        IPP.append(PPI)
        zl=zl+(zstep)


    zl=ZLPP[IPP.index(max(IPP))]


    plt.plot(ZLPP,IPP)
    plt.show()

    #points=100
    #xv,yv=np.meshgrid(np.linspace(-20,20,points),np.linspace(-20,20,points))
    #iv=TestInt.get(xv,yv)
    #ax.plot_surface(xv,yv,iv,alpha=0.5)
    plt.show()
coord=(xl,yl,zl)
robot.MoveJ(target.Pose()*transl(coord))

E=np.sqrt((Ix-xl)**2+(Iy-yl)**2)
print('***Linear Translation********************************************************')
print(Ldata)
print('_________SSAP Report:_________')
print('Calculated peak is at',xl,yl)
print('True peak is at',Ix,Iy)
print('Error is:',E)
print('Linear step size is:',step)

--- Python program Set Target Pos ---
from robolink import *
from robodk import *
RDK = Robolink()

# Get a reference to the target object
PR = RDK.Item('Photo Resistor',ITEM_TYPE_TARGET)
CT= RDK.Item('Crystal Target',ITEM_TYPE_TARGET)
TPP= RDK.Item('TPP',ITEM_TYPE_TARGET)

# Define the new position and orientation of the frame

x=0
y=0
z=-8*25.4

PR.setPose(Pose(x,y,z,0,0,0))
CT.setPose(Pose(x,y,z/2,0,0,0))
TPP.setPose(Pose(x-1000,y,z/2,0,90,0))


reference = TPP.Parent()
print("Target attached to: " + reference.Name())

# You can also move this target to a new reference:
#target.setParent(new_frame)

--- Python program Hexagon Test ---
# Draw a hexagon around the current robot position

from robodk.robolink import *  # RoboDK's API
from robodk.robomath import *  # Robot toolbox

# Start the RoboDK API:
RDK = Robolink()

# Get the robot (first robot found):

robot = RDK.Item('Mecademic Meca500 R3')     # retrieve the robot by name

# Get the reference target by name:

tool=RDK.Item('CrystalToolSample')
robot.setPoseTool(tool) # Update the TCP
target = RDK.Item('TPP')
target_pose = target.Pose()
robot.MoveJ(target)

target_pose = robot.Pose()
xyz_ref = target_pose.Pos()

# Move the robot to the reference point (current position/redundant):
robot.MoveJ(target_pose)

# Draw a hexagon around the reference target:
for i in range(7):
    ang = i * 2 * pi / 6  # Angle = 0,60,120,...,360
    R = 20  # Polygon radius

    # Calculate the new position around the reference:
    x = xyz_ref[0] + R * cos(ang)  # new X coordinate
    z = xyz_ref[1] + R * sin(ang)  # new Y coordinate
    y = xyz_ref[2]  # new Z coordinate
    target_pose.setPos([x, y, z])

    # Move to the new target:
    robot.MoveL(target_pose)

# Trigger a program call at the end of the movement
robot.RunInstruction('Program_Done')

# Move back to the reference target:
robot.MoveL(target_pose)

--- Python program Prog12 ---
from robolink import *  # import the RoboDK API
from robodk import *  # import the RoboDK API for robots

# Connect to the RoboDK API
RDK = Robolink()

# Get the robot item from the RoboDK station
robot = RDK.Item('Mecademic Meca500 R3')

# Get the tool item from the RoboDK station
tool = RDK.Item('CrystalToolSample')

# Get the reference item from the RoboDK station
reference = RDK.Item('LED')

# Set the tool and reference frames for the robot
robot.setPoseTool(tool.Pose())
robot.setPoseFrame(reference.Pose())

# Define the start and end positions for the translation
start_pos = [0, 0, 0.2]  # in meters
end_pos = [0, 0.1, 0.2]  # in meters

# Define the speed and acceleration for the robot movement
speed = 50  # in mm/s
accel = 100  # in mm/s^2

# Create a linear movement instruction for the robot
move_instr = robot.MoveL(  # Move in a straight line
    pose_transl(start_pos),  # Start position
    pose_transl(end_pos),  # End position
    speed,  # Movement speed
    accel  # Movement acceleration
)

# Simulate the robot movement in RoboDK
robot.Simulate()

# Generate the robot program for the linear movement instruction
program = move_instr.Program()

# Send the program to the robot controller for execution
robot.SendProgram(program)

--- Python program Prog13 ---
from robolink import *  # import the RoboDK API
from robodk import *  # import the RoboDK API for robots

# Connect to the RoboDK API
RDK = Robolink()

# Get the robot item from the RoboDK station
robot = RDK.Item('Mecademic Meca500 R3')

# Get the tool item from the RoboDK station
tool = RDK.Item('CrystalToolSample')

# Get the reference item from the RoboDK station
reference = RDK.Item('LED')

# Set the tool and reference frames for the robot
robot.setPoseTool(tool.Pose())
robot.setPoseFrame(reference.Pose())

# Define the start and end positions for the translation
start_pos = [0, 0, 0.2]  # in meters
end_pos = [0, 0.1, 0.2]  # in meters

# Define the speed and acceleration for the robot movement
speed = 50  # in mm/s
accel = 100  # in mm/s^2

# Create a linear movement instruction for the robot
robot.MoveL(transl*(start_pos))
